FUNCTION F_TzInfoBiasToTzStr : STRING
VAR_INPUT
	tzBias : DINT;
END_VAR
VAR
	UtcOffset : DINT;
END_VAR

UtcOffset := (0-tzBias) / 60;
IF UtcOffset > 0 AND UtcOffset < 10 THEN
	F_TzInfoBiasToTzStr := CONCAT(STR1:= 'UTC+0', STR2:= DINT_TO_STRING(UtcOffset));
ELSIF UtcOffset >= 10 AND UtcOffset <= 12 THEN
	F_TzInfoBiasToTzStr := CONCAT(STR1:= 'UTC+', STR2:= DINT_TO_STRING(UtcOffset));
ELSIF UtcOffset < 0 AND UtcOffset > -10 THEN
	F_TzInfoBiasToTzStr := CONCAT(STR1:= 'UTC-0', STR2:= DINT_TO_STRING(UtcOffset));
ELSIF UtcOffset <=10 AND UtcOffset >= -12 THEN
	F_TzInfoBiasToTzStr := CONCAT(STR1:= 'UTC-', STR2:= DINT_TO_STRING(UtcOffset));
ELSIF UtcOffset = 0 THEN
	F_TzInfoBiasToTzStr := 'UTC';
END_IF

END_FUNCTION

(* stored: Version 1.1.0.1, ProductVersion 3.1.4024.12
   POU F_TzInfoBiasToTzStr: Id {dd259556-d823-4140-8529-19652193adfd}, SpecialFunc None *)
